SUBAPPLICATION FBs9 (* Subapplication Type *)
  (* Standard: 61499-2 *)
  (* Version 1.0, 2025-05-03, cochicde *)
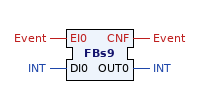
  EVENT_INPUT
    EI0;
  END_EVENT
  EVENT_OUTPUT
    CNF;
  END_EVENT
  VAR_INPUT
    DI0 : INT;
  END_VAR
  VAR_OUTPUT
    OUT0 : INT;
  END_VAR
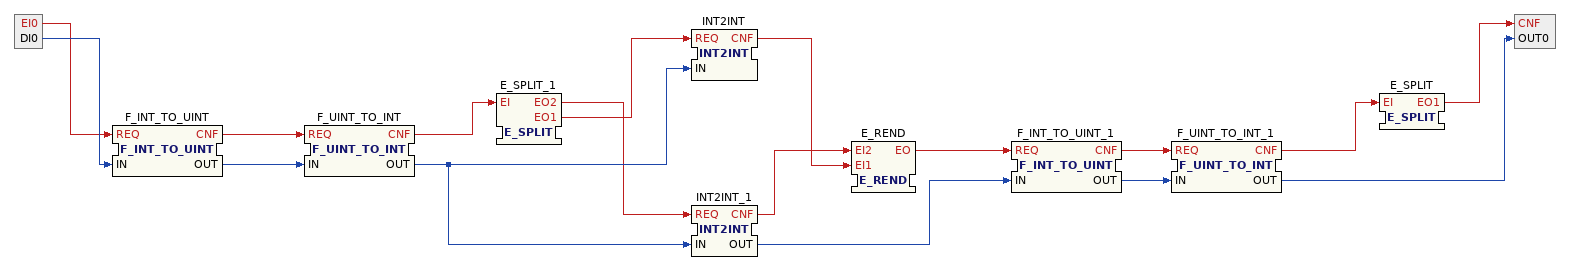
  FBS
    F_UINT_TO_INT : F_UINT_TO_INT;
    INT2INT_1 : INT2INT;
    E_SPLIT_1 : E_SPLIT;
    INT2INT : INT2INT;
    F_INT_TO_UINT : F_INT_TO_UINT;
    F_INT_TO_UINT_1 : F_INT_TO_UINT;
    F_UINT_TO_INT_1 : F_UINT_TO_INT;
    E_REND : E_REND;
    E_SPLIT : E_SPLIT;
  END_FBS
  EVENT_CONNECTIONS
    F_INT_TO_UINT.CNF TO F_UINT_TO_INT.REQ;
    F_UINT_TO_INT.CNF TO E_SPLIT_1.EI;
    E_SPLIT_1.EO2 TO INT2INT_1.REQ;
    INT2INT_1.CNF TO E_REND.EI2;
    E_SPLIT_1.EO1 TO INT2INT.REQ;
    INT2INT.CNF TO E_REND.EI1;
    F_UINT_TO_INT_1.CNF TO E_SPLIT.EI;
    E_REND.EO TO F_INT_TO_UINT_1.REQ;
    F_INT_TO_UINT_1.CNF TO F_UINT_TO_INT_1.REQ;
    EI0 TO F_INT_TO_UINT.REQ;
    E_SPLIT.EO1 TO CNF;
  END_CONNECTIONS
  DATA_CONNECTIONS
    F_INT_TO_UINT.OUT TO F_UINT_TO_INT.IN;
    F_UINT_TO_INT.OUT TO INT2INT.IN;
    F_UINT_TO_INT.OUT TO INT2INT_1.IN;
    INT2INT_1.OUT TO F_INT_TO_UINT_1.IN;
    F_INT_TO_UINT_1.OUT TO F_UINT_TO_INT_1.IN;
    DI0 TO F_INT_TO_UINT.IN;
    F_UINT_TO_INT_1.OUT TO OUT0;
  END_CONNECTIONS
END_SUBAPPLICATION
